FUNCTION_BLOCK CentralController (* Basic Function Block Type *)
  (* Standard: 61499-2 *)
  (* Version 0.0, 2011-08-30, cspgen, nxtControl GmbH, Template *)
  PACKAGE Main;
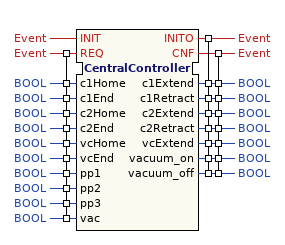
  EVENT_INPUT
    INIT; (* Initialization Request *)
    REQ WITH c1Home, c1End, c2Home, c2End, vcHome, vcEnd, pp1, pp2, pp3, vac; (* REQ *)
  END_EVENT
  EVENT_OUTPUT
    INITO WITH c1Extend, c1Retract, c2Extend, c2Retract, vcExtend, vacuum_on, vacuum_off; (* INITO *)
    CNF WITH c1Extend, c1Retract, c2Extend, c2Retract, vcExtend, vacuum_on, vacuum_off; (* CNF *)
  END_EVENT
  VAR_INPUT
    c1Home : BOOL;
    c1End : BOOL;
    c2Home : BOOL;
    c2End : BOOL;
    vcHome : BOOL;
    vcEnd : BOOL;
    pp1 : BOOL;
    pp2 : BOOL;
    pp3 : BOOL;
    vac : BOOL;
  END_VAR
  VAR_OUTPUT
    c1Extend : BOOL;
    c1Retract : BOOL;
    c2Extend : BOOL;
    c2Retract : BOOL;
    vcExtend : BOOL;
    vacuum_on : BOOL;
    vacuum_off : BOOL;
  END_VAR
  EC_STATES
    START; (* Initial State *)
    INIT : INIT -> INITO; (* Initialization *)
    s_0 : a_0000000_0000000;
    s_1 : a_0010000_1010010_CNF -> CNF;
    s_2 : a_1010000_1010010_CNF -> CNF;
    s_3 : a_1000000_1010010_CNF -> CNF;
    s_4 : a_0000100_1111011_CNF -> CNF;
    s_5 : a_0000110_1111110_CNF -> CNF;
    s_6 : a_0101000_0101011_CNF -> CNF;
    s_7 : a_0000101_0111100_CNF -> CNF;
  END_STATES
  EC_TRANSITIONS
    START TO INIT := INIT;
    INIT TO s_0 := 1;
    s_0 TO s_1 := REQ&pp2;
    s_0 TO s_3 := REQ&pp1;
    s_0 TO s_2 := REQ&pp3;
    s_1 TO s_4 := REQ&c2End;
    s_2 TO s_4 := REQ&c2End;
    s_3 TO s_4 := REQ&c1End;
    s_4 TO s_5 := REQ&((NOT  (vac)) AND (vcEnd));
    s_4 TO s_6 := REQ&((vcHome) AND (vac));
    s_4 TO s_3 := REQ&((c1Home) AND (((vcHome) AND (pp1))));
    s_4 TO s_1 := REQ&((((c1Home) AND (c2Home))) AND (vcHome));
    s_5 TO s_4 := REQ&((c1End) OR (c2End));
    s_5 TO s_7 := REQ&vcEnd;
    s_6 TO s_1 := REQ&((((NOT  (((pp1) OR (vac)))) AND (vcHome))) AND (pp2));
    s_6 TO s_2 := REQ&((((NOT  (vac)) AND (vcHome))) AND (pp3));
    s_6 TO s_5 := REQ&((((c2Home) AND (vac))) AND (c1Home));
    s_6 TO s_3 := REQ&((c2Home) AND (((vcHome) AND (pp1))));
    s_7 TO s_4 := REQ&((((NOT  (pp1)) AND (pp2))) OR (((pp1) AND (pp3))));
    s_7 TO s_6 := REQ&c2Home;
  END_TRANSITIONS
  ALGORITHM INIT IN ST: (* Initialization algorithm *)
REQ := FALSE;
c1Extend:=FALSE;
c1Retract:=FALSE;
c2Extend:=FALSE;
c2Retract:=FALSE;
vcExtend:=FALSE;
vacuum_on:=FALSE;
vacuum_off:=FALSE;
  END_ALGORITHM
  ALGORITHM a_0000100_1111011_CNF IN ST:
 REQ := FALSE;
IF c1Extend THEN
c1Extend := TRUE;
ELSE
c1Extend := FALSE;
END_IF;
IF c1Retract THEN
c1Retract := TRUE;
ELSE
c1Retract := FALSE;
END_IF;
IF c2Extend THEN
c2Extend := TRUE;
ELSE
c2Extend := FALSE;
END_IF;
IF c2Retract THEN
c2Retract := TRUE;
ELSE
c2Retract := FALSE;
END_IF;
IF vcExtend THEN
vcExtend := FALSE;
ELSE
vcExtend := TRUE;
END_IF;
IF vacuum_on THEN
vacuum_on := TRUE;
ELSE
vacuum_on := FALSE;
END_IF;
IF vacuum_off THEN
vacuum_off := TRUE;
ELSE
vacuum_off := FALSE;
END_IF;
  END_ALGORITHM
  ALGORITHM a_0000000_0000000 IN ST:
 REQ := FALSE;
IF c1Extend THEN
c1Extend := FALSE;
ELSE
c1Extend := FALSE;
END_IF;
IF c1Retract THEN
c1Retract := FALSE;
ELSE
c1Retract := FALSE;
END_IF;
IF c2Extend THEN
c2Extend := FALSE;
ELSE
c2Extend := FALSE;
END_IF;
IF c2Retract THEN
c2Retract := FALSE;
ELSE
c2Retract := FALSE;
END_IF;
IF vcExtend THEN
vcExtend := FALSE;
ELSE
vcExtend := FALSE;
END_IF;
IF vacuum_on THEN
vacuum_on := FALSE;
ELSE
vacuum_on := FALSE;
END_IF;
IF vacuum_off THEN
vacuum_off := FALSE;
ELSE
vacuum_off := FALSE;
END_IF;
  END_ALGORITHM
  ALGORITHM a_1010000_1010010_CNF IN ST:
 REQ := FALSE;
IF c1Extend THEN
c1Extend := TRUE;
ELSE
c1Extend := TRUE;
END_IF;
IF c1Retract THEN
c1Retract := FALSE;
ELSE
c1Retract := FALSE;
END_IF;
IF c2Extend THEN
c2Extend := TRUE;
ELSE
c2Extend := TRUE;
END_IF;
IF c2Retract THEN
c2Retract := FALSE;
ELSE
c2Retract := FALSE;
END_IF;
IF vcExtend THEN
vcExtend := FALSE;
ELSE
vcExtend := FALSE;
END_IF;
IF vacuum_on THEN
vacuum_on := TRUE;
ELSE
vacuum_on := FALSE;
END_IF;
IF vacuum_off THEN
vacuum_off := FALSE;
ELSE
vacuum_off := FALSE;
END_IF;
  END_ALGORITHM
  ALGORITHM a_0010000_1010010_CNF IN ST:
 REQ := FALSE;
IF c1Extend THEN
c1Extend := TRUE;
ELSE
c1Extend := FALSE;
END_IF;
IF c1Retract THEN
c1Retract := FALSE;
ELSE
c1Retract := FALSE;
END_IF;
IF c2Extend THEN
c2Extend := TRUE;
ELSE
c2Extend := TRUE;
END_IF;
IF c2Retract THEN
c2Retract := FALSE;
ELSE
c2Retract := FALSE;
END_IF;
IF vcExtend THEN
vcExtend := FALSE;
ELSE
vcExtend := FALSE;
END_IF;
IF vacuum_on THEN
vacuum_on := TRUE;
ELSE
vacuum_on := FALSE;
END_IF;
IF vacuum_off THEN
vacuum_off := FALSE;
ELSE
vacuum_off := FALSE;
END_IF;
  END_ALGORITHM
  ALGORITHM a_1000000_1010010_CNF IN ST:
 REQ := FALSE;
IF c1Extend THEN
c1Extend := TRUE;
ELSE
c1Extend := TRUE;
END_IF;
IF c1Retract THEN
c1Retract := FALSE;
ELSE
c1Retract := FALSE;
END_IF;
IF c2Extend THEN
c2Extend := TRUE;
ELSE
c2Extend := FALSE;
END_IF;
IF c2Retract THEN
c2Retract := FALSE;
ELSE
c2Retract := FALSE;
END_IF;
IF vcExtend THEN
vcExtend := FALSE;
ELSE
vcExtend := FALSE;
END_IF;
IF vacuum_on THEN
vacuum_on := TRUE;
ELSE
vacuum_on := FALSE;
END_IF;
IF vacuum_off THEN
vacuum_off := FALSE;
ELSE
vacuum_off := FALSE;
END_IF;
  END_ALGORITHM
  ALGORITHM a_0000110_1111110_CNF IN ST:
 REQ := FALSE;
IF c1Extend THEN
c1Extend := TRUE;
ELSE
c1Extend := FALSE;
END_IF;
IF c1Retract THEN
c1Retract := TRUE;
ELSE
c1Retract := FALSE;
END_IF;
IF c2Extend THEN
c2Extend := TRUE;
ELSE
c2Extend := FALSE;
END_IF;
IF c2Retract THEN
c2Retract := TRUE;
ELSE
c2Retract := FALSE;
END_IF;
IF vcExtend THEN
vcExtend := TRUE;
ELSE
vcExtend := TRUE;
END_IF;
IF vacuum_on THEN
vacuum_on := TRUE;
ELSE
vacuum_on := TRUE;
END_IF;
IF vacuum_off THEN
vacuum_off := FALSE;
ELSE
vacuum_off := FALSE;
END_IF;
  END_ALGORITHM
  ALGORITHM a_0101000_0101011_CNF IN ST:
 REQ := FALSE;
IF c1Extend THEN
c1Extend := FALSE;
ELSE
c1Extend := FALSE;
END_IF;
IF c1Retract THEN
c1Retract := TRUE;
ELSE
c1Retract := TRUE;
END_IF;
IF c2Extend THEN
c2Extend := FALSE;
ELSE
c2Extend := FALSE;
END_IF;
IF c2Retract THEN
c2Retract := TRUE;
ELSE
c2Retract := TRUE;
END_IF;
IF vcExtend THEN
vcExtend := FALSE;
ELSE
vcExtend := FALSE;
END_IF;
IF vacuum_on THEN
vacuum_on := TRUE;
ELSE
vacuum_on := FALSE;
END_IF;
IF vacuum_off THEN
vacuum_off := TRUE;
ELSE
vacuum_off := FALSE;
END_IF;
  END_ALGORITHM
  ALGORITHM a_0000101_0111100_CNF IN ST:
 REQ := FALSE;
IF c1Extend THEN
c1Extend := FALSE;
ELSE
c1Extend := FALSE;
END_IF;
IF c1Retract THEN
c1Retract := TRUE;
ELSE
c1Retract := FALSE;
END_IF;
IF c2Extend THEN
c2Extend := TRUE;
ELSE
c2Extend := FALSE;
END_IF;
IF c2Retract THEN
c2Retract := TRUE;
ELSE
c2Retract := FALSE;
END_IF;
IF vcExtend THEN
vcExtend := TRUE;
ELSE
vcExtend := TRUE;
END_IF;
IF vacuum_on THEN
vacuum_on := FALSE;
ELSE
vacuum_on := FALSE;
END_IF;
IF vacuum_off THEN
vacuum_off := FALSE;
ELSE
vacuum_off := TRUE;
END_IF;
  END_ALGORITHM
END_FUNCTION_BLOCK
